(* IEC 61131-3 sources: volt/packages/volt-lsp-iec/test-corpus/bakon-nano/Device/Plc Logic/Application/Library Manager/SysTimeRtc, 23 files *)

(* ---- RTS_SYSTIMEDATE.dut ---- *)
TYPE RTS_SYSTIMEDATE :
STRUCT
	WYEAR : UINT;
	WMONTH : UINT;
	WDAY : UINT;
	WHOUR : UINT;
	WMINUTE : UINT;
	WSECOND : UINT;
	WMILLISECONDS : UINT;
	WDAYOFWEEK : UINT;
	WYDAY : UINT;
END_STRUCT
END_TYPE

(* ---- SYSTIMEDATE.dut ---- *)
TYPE SYSTIMEDATE : RTS_SYSTIMEDATE;
END_TYPE

(* ---- TIMEZONEINFORMATION.dut ---- *)
TYPE TIMEZONEINFORMATION :
STRUCT
	ULSTANDARDDATE : UDINT;
	ULDAYLIGHTDATE : UDINT;
	SZSTANDARDNAME : STRING(32);
	SZDAYLIGHTNAME : STRING(32);
	IBIAS : INT;
	ISTANDARDBIAS : INT;
	IDAYLIGHTBIAS : INT;
END_STRUCT
END_TYPE

(* ---- TIMEZONEINFORMATION2.dut ---- *)
TYPE TIMEZONEINFORMATION2 :
STRUCT
	UTCOFFSETSECONDS : DINT;
	ISDST : DINT;
	SZTIMEZONE : STRING(127);
END_STRUCT
END_TYPE

(* ---- GVL.gvl ---- *)
VAR_GLOBAL
	RTC_12HOURS : DINT := 0;
	RTC_24HOURS : DINT := 1;
	RTC_BATTERY_FAILED : DINT := 0;
	RTC_BATTERY_OK : DINT := 1;
	RTC_CTRL_CHECKBATTERY : DWORD := 0;
	RTC_CTRL_HOURMODE : DWORD := 1;
END_VAR

(* ---- SYSTIMEGETDATE.pou ---- *)
FUNCTION SYSTIMEGETDATE : UDINT
VAR_IN_OUT
	TIMEDATE : SYSTIMEDATE;
END_VAR
END_FUNCTION

(* ---- SYSTIMEGETTIMESTAMP.pou ---- *)
FUNCTION SYSTIMEGETTIMESTAMP : UDINT
END_FUNCTION

(* ---- SYSTIMERTCCONTROL.pou ---- *)
FUNCTION SYSTIMERTCCONTROL : RTS_IEC_RESULT
VAR_INPUT
	ICONTROLTAG : DINT;
END_VAR
VAR_IN_OUT
	PDICONTROLRESULT : DINT;
END_VAR
END_FUNCTION

(* ---- SYSTIMERTCCONVERTDATETOHIGHRES.pou ---- *)
FUNCTION SYSTIMERTCCONVERTDATETOHIGHRES : RTS_IEC_RESULT
VAR_IN_OUT
	PDATE : SYSTIMEDATE;
	PTIMESTAMP : SYSTIME;
END_VAR
END_FUNCTION

(* ---- SYSTIMERTCCONVERTDATETOUTC.pou ---- *)
FUNCTION SYSTIMERTCCONVERTDATETOUTC : RTS_IEC_RESULT
VAR_IN_OUT
	PDATE : SYSTIMEDATE;
	PDWTIMESTAMPUTC : DWORD;
END_VAR
END_FUNCTION

(* ---- SYSTIMERTCCONVERTHIGHRESTODATE.pou ---- *)
FUNCTION SYSTIMERTCCONVERTHIGHRESTODATE : RTS_IEC_RESULT
VAR_IN_OUT
	PTIMESTAMP : SYSTIME;
	PDATE : SYSTIMEDATE;
END_VAR
END_FUNCTION

(* ---- SYSTIMERTCCONVERTHIGHRESTOLOCAL.pou ---- *)
FUNCTION SYSTIMERTCCONVERTHIGHRESTOLOCAL : RTS_IEC_RESULT
VAR_IN_OUT
	PTIMESTAMP : SYSTIME;
	PDATE : SYSTIMEDATE;
END_VAR
END_FUNCTION

(* ---- SYSTIMERTCCONVERTLOCALTOHIGHRES.pou ---- *)
FUNCTION SYSTIMERTCCONVERTLOCALTOHIGHRES : RTS_IEC_RESULT
VAR_IN_OUT
	PDATE : SYSTIMEDATE;
	PTIMESTAMP : SYSTIME;
END_VAR
END_FUNCTION

(* ---- SYSTIMERTCCONVERTLOCALTOUTC.pou ---- *)
FUNCTION SYSTIMERTCCONVERTLOCALTOUTC : RTS_IEC_RESULT
VAR_INPUT
	DWTIMESTAMPLOCAL : DWORD;
END_VAR
VAR_IN_OUT
	PDWTIMESTAMPUTC : DWORD;
END_VAR
END_FUNCTION

(* ---- SYSTIMERTCCONVERTUTCTODATE.pou ---- *)
FUNCTION SYSTIMERTCCONVERTUTCTODATE : RTS_IEC_RESULT
VAR_INPUT
	DWTIMESTAMPUTC : DWORD;
END_VAR
VAR_IN_OUT
	PDATE : SYSTIMEDATE;
END_VAR
END_FUNCTION

(* ---- SYSTIMERTCCONVERTUTCTOLOCAL.pou ---- *)
FUNCTION SYSTIMERTCCONVERTUTCTOLOCAL : RTS_IEC_RESULT
VAR_INPUT
	DWTIMESTAMPUTC : DWORD;
END_VAR
VAR_IN_OUT
	PDWTIMESTAMPLOCAL : DWORD;
END_VAR
END_FUNCTION

(* ---- SYSTIMERTCGET.pou ---- *)
FUNCTION SYSTIMERTCGET : DWORD
VAR_IN_OUT
	PRESULT : RTS_IEC_RESULT;
END_VAR
END_FUNCTION

(* ---- SYSTIMERTCGETTIMEZONE.pou ---- *)
FUNCTION SYSTIMERTCGETTIMEZONE : RTS_IEC_RESULT
VAR_IN_OUT
	PTIMEZONE : TimezoneInformation;
END_VAR
END_FUNCTION

(* ---- SYSTIMERTCGETTIMEZONE2.pou ---- *)
FUNCTION SYSTIMERTCGETTIMEZONE2 : RTS_IEC_RESULT
VAR_IN_OUT
	PTZI : TimezoneInformation2;
END_VAR
END_FUNCTION

(* ---- SYSTIMERTCHIGHRESGET.pou ---- *)
FUNCTION SYSTIMERTCHIGHRESGET : RTS_IEC_RESULT
VAR_IN_OUT
	PTIMESTAMP : SYSTIME;
END_VAR
END_FUNCTION

(* ---- SYSTIMERTCHIGHRESSET.pou ---- *)
FUNCTION SYSTIMERTCHIGHRESSET : RTS_IEC_RESULT
VAR_IN_OUT
	PTIMESTAMP : SYSTIME;
END_VAR
END_FUNCTION

(* ---- SYSTIMERTCSET.pou ---- *)
FUNCTION SYSTIMERTCSET : RTS_IEC_RESULT
VAR_INPUT
	ULTIMESTAMP : DWORD;
END_VAR
END_FUNCTION

(* ---- SYSTIMERTCSETTIMEZONE.pou ---- *)
FUNCTION SYSTIMERTCSETTIMEZONE : RTS_IEC_RESULT
VAR_IN_OUT
	PTIMEZONE : TimezoneInformation;
END_VAR
END_FUNCTION
